(* CODESYS project BlowerMotor.xml

Project tree, tasks and I/O mapping:
  function block BlowerMotor [LD]
*)

// BlowerMotor
FUNCTION_BLOCK BlowerMotor
//  .					.					.
VAR_INPUT
	Run: 				BOOL;				//
	Override: 			BOOL;				//
	OverrideMotor: 		BOOL;				//
END_VAR
VAR_OUTPUT
	MotorOutput: 		BOOL;				//
END_VAR
VAR
END_VAR

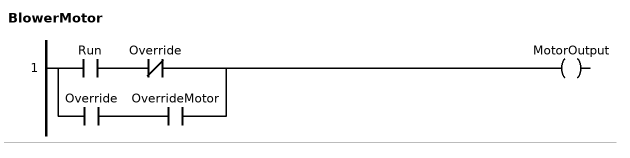
// NETWORK 1
MotorOutput := Run AND NOT Override OR Override AND OverrideMotor;

END_FUNCTION_BLOCK
